TYPE ST_APP_INFO :
STRUCT
  AppInit           : E_PROGRESS;
  Instance          : E_INSTANCE;  // process ID from which the MoverPerMinute counter is copied
  MoverPerMinute    : UDINT;
  MoverTotal        : UDINT;
  StationParameterVariant : UDINT;
END_STRUCT
END_TYPE

(* stored: Version 1.1.0.1
   DUT ST_APP_INFO: Id {52e2dffe-3040-4a6f-ad8d-633ed2701922} *)
